(*
SPDX-FileCopyrightText: © 2026 Oleksandr Tiutyk <trofimich@gmail.com>
SPDX-License-Identifier: MIT
License: https://opensource.org/license/mit
*)

INTERFACE IWhileActivity EXTENDS ISequenceActivity

{attribute 'monitoring' := 'call'}
PROPERTY Condition : ICondition
GET
END_GET
SET
END_SET
END_PROPERTY

METHOD Configure
VAR_INPUT
	condition : ICondition; 
END_VAR
END_METHOD

END_INTERFACE

(* stored: Version 1.1.0.1
   Itf IWhileActivity: Id {48afd1de-38c9-486e-a527-23b68379f379}
   Property Condition: Id {121e9e17-db69-4d58-a344-e6e8a3a42d4b}
   Get Get: Id {9c48afd2-d45d-4366-84e1-f61bd2c6adc9}
   Set Set: Id {28ceb78b-c399-40fd-b3cc-862dfac65f1c}
   Method Configure: Id {1073bb11-2516-4e4a-b056-d98e3143c9fd} *)
